PROGRAM MAIN
VAR
	A1: Achse1;
END_VAR

A1();

END_PROGRAM

(* stored: Version 1.1.0.1, ProductVersion 3.1.4024.4
   POU MAIN: Id {8c3fea05-08d9-4bdc-b5eb-0bd792ace699}, SpecialFunc None *)
